SUBAPPLICATION DDS_SERVER (* Wrapper for DDS Publisher and Subscriber Pair as a Client *)
  (* Standard: 61499-2 *)
  (* Version 1.0, 2023-03-15, Tim Hesse *)
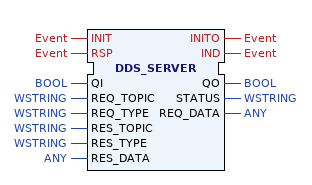
  EVENT_INPUT
    INIT; (* Initialization Request *)
    RSP; (* Application Response to IND *)
  END_EVENT
  EVENT_OUTPUT
    INITO; (* Initialization Confirm *)
    IND; (* Confirmation of Requested Service *)
  END_EVENT
  VAR_INPUT
    QI : BOOL; (* Input event qualifier *)
    REQ_TOPIC : WSTRING; (* Request DDS Topic *)
    REQ_TYPE : WSTRING; (* Request DDS Type *)
    RES_TOPIC : WSTRING; (* Response DDS Topic *)
    RES_TYPE : WSTRING; (* Response DDS Type *)
    RES_DATA : ANY; (* Response Data *)
  END_VAR
  VAR_OUTPUT
    QO : BOOL; (* Output event qualifier *)
    STATUS : WSTRING; (* Service Status *)
    REQ_DATA : ANY; (* Request Data *)
  END_VAR
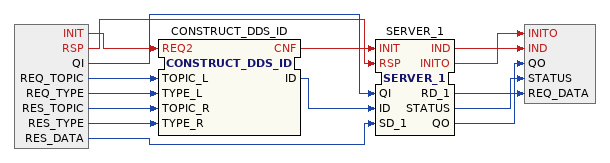
  FBS
    CONSTRUCT_DDS_ID : CONSTRUCT_DDS_ID;
    SERVER_1 : SERVER_1;
  END_FBS
  EVENT_CONNECTIONS
    INIT TO CONSTRUCT_DDS_ID.REQ2;
    CONSTRUCT_DDS_ID.CNF TO SERVER_1.INIT;
    RSP TO SERVER_1.RSP;
    SERVER_1.IND TO IND;
    SERVER_1.INITO TO INITO;
  END_CONNECTIONS
  DATA_CONNECTIONS
    REQ_TOPIC TO CONSTRUCT_DDS_ID.TOPIC_L;
    REQ_TYPE TO CONSTRUCT_DDS_ID.TYPE_L;
    RES_TOPIC TO CONSTRUCT_DDS_ID.TOPIC_R;
    RES_TYPE TO CONSTRUCT_DDS_ID.TYPE_R;
    QI TO SERVER_1.QI;
    CONSTRUCT_DDS_ID.ID TO SERVER_1.ID;
    RES_DATA TO SERVER_1.SD_1;
    SERVER_1.RD_1 TO REQ_DATA;
    SERVER_1.STATUS TO STATUS;
    SERVER_1.QO TO QO;
  END_CONNECTIONS
END_SUBAPPLICATION
